// TIA Portal V20 export
// export: Created 2026-04-11T06:02:30.1321665Z, ExportSetting WithDefaults, DisplayName Totally Integrated Automation Portal, DisplayVersion V20, DisplayName TIA Portal Openness, DisplayVersion V20, DisplayName TIA Portal Version Control Interface, DisplayVersion V20, DisplayName STEP 7 Professional, DisplayVersion V20, DisplayName STEP 7 Safety, DisplayVersion V20, DisplayName WinCC Basic/Comfort/Advanced, DisplayVersion V20, DisplayName WinCC Unified, DisplayVersion V20
TYPE "udtError_Brabender"
// stored: IsFailsafeCompliant false
   STRUCT
      LoadCellSignal { ExternalWritable := 'False'} : Bool;   // Load cell signal
      RefillFault { ExternalWritable := 'False'} : Bool;   // Refill fault
      Underload { ExternalWritable := 'False'} : Bool;   // Underload
      Overload { ExternalWritable := 'False'} : Bool;   // Overload
      ControlDiffNeg { ExternalWritable := 'False'} : Bool;   // Control difference -
      ControlDiffPos { ExternalWritable := 'False'} : Bool;   // Control difference +
      SpeedMin { ExternalWritable := 'False'} : Bool;   // Speed minimum
      SpeedMax { ExternalWritable := 'False'} : Bool;   // Speed maximum
      MemoryModuleError { ExternalWritable := 'False'} : Bool;   // Memory module error
      AutoTareError { ExternalWritable := 'False'} : Bool;   // Auto-tare error
      SoftStartError { ExternalWritable := 'False'} : Bool;   // Soft start error
      AV_Error { ExternalWritable := 'False'} : Bool;   // AV error
      CM_Error { ExternalWritable := 'False'} : Bool;   // CM error
      FC_Error { ExternalWritable := 'False'} : Bool;   // FC error
      CoriolisSpeed { ExternalWritable := 'False'} : Bool;   // Coriolis speed
      CommunicationError { ExternalWritable := 'False'} : Bool;   // Communication error ISC/CB
      IO_Error { ExternalWritable := 'False'} : Bool;   // IO error
      FaultExtern { ExternalWritable := 'False'} : Bool;   // Fault extern
      Overpressure { ExternalWritable := 'False'} : Bool;   // Overpressure
      BeltRun { ExternalWritable := 'False'} : Bool;   // Belt run
      ExtWarning { ExternalWritable := 'False'} : Bool;   // Ext. warning
      GeneralError { ExternalWritable := 'False'} : Bool;   // General error, see Brabender HMI
      StartTimeOut { ExternalWritable := 'False'} : Bool;   // If start is requested, but started status does not come
      LocalDisconnect { ExternalWritable := 'False'} : Bool;   // Local Disconnect is Off
   END_STRUCT;
END_TYPE
